// TIA Portal V20 export
DATA_BLOCK "DB_DataPositions"   // DB701
{ S7_Optimized_Access := 'TRUE' }
// stored: AutoNumber false, MemoryReserve 100
   VAR
      Position : Array[0..52] of "UDT_Tracability";
   END_VAR
BEGIN
END_DATA_BLOCK
